FUNCTION_BLOCK L2_ASetupRSPHDLR (* Basic Function Block Type *)
  (* Standard: 61499-2 *)
  (* Version 0.0, 2014-11-28, EQUEROL, UJI *)
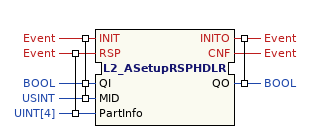
  EVENT_INPUT
    INIT WITH QI, MID; (* Initialization Request *)
    RSP WITH PartInfo; (* Normal Execution Request *)
  END_EVENT
  EVENT_OUTPUT
    INITO WITH QO; (* Initialization Confirm *)
    CNF; (* Execution Confirmation *)
  END_EVENT
  VAR_INPUT
    QI : BOOL; (* Input event qualifier *)
    MID : USINT; (* Machine identifier *)
    PartInfo : ARRAY [0..3] OF UINT; (* ID, Family, Type, MID *)
  END_VAR
  VAR_OUTPUT
    QO : BOOL; (* Output event qualifier *)
  END_VAR
  VAR
    Accepted : BOOL := FALSE; (* This variable allow to diferentiate between accepted and rejected request *)
  END_VAR
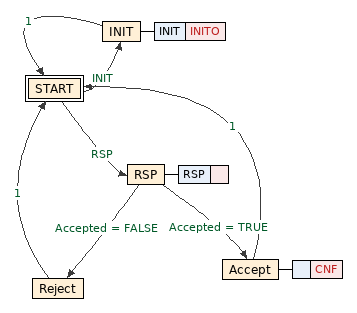
  EC_STATES
    START; (* Initial State *)
    INIT : INIT -> INITO; (* Initialization *)
    RSP : RSP; (* Normal execution *)
    Accept : -> CNF;
    Reject;
  END_STATES
  EC_TRANSITIONS
    START TO INIT := INIT;
    INIT TO START := 1;
    START TO RSP := RSP;
    RSP TO Accept := Accepted = TRUE;
    Accept TO START := 1;
    Reject TO START := 1;
    RSP TO Reject := Accepted = FALSE;
  END_TRANSITIONS
  ALGORITHM INIT IN ST: (* Initialization algorithm *)
QO := QI;
  END_ALGORITHM
  ALGORITHM RSP IN ST: (* Normally executed algorithm *)
IF MID = PartInfo[3] THEN
	Accepted := TRUE;
ELSE
	Accepted := FALSE;
END_IF;
  END_ALGORITHM
END_FUNCTION_BLOCK
